TYPE E_EcSystemStatus :
(

	eEcSystem_Start							:= 0,
	eEcSystem_ReadConfSystem

);
END_TYPE
(* End *)

(* stored: Version 1.1.0.1, ProductVersion 3.1.4022.12
   DUT E_EcSystemStatus: Id {a178aca6-8aba-42c4-a916-dc9d26ffd7e2} *)
